// TIA Portal V18 export
// export: Created 2026-03-12T16:04:34.7244026Z, ExportSetting WithDefaults, DisplayName Totally Integrated Automation Portal, DisplayVersion V18 Update 5, DisplayName TIA Portal Openness, DisplayVersion V18 Update 5, DisplayName TIA Portal Version Control Interface, DisplayVersion V18, DisplayName SINAMICS Startdrive Advanced, DisplayVersion V18, DisplayName SINAMICS Startdrive G130, G150, S120, S150, SINAMICS MV, S210, DisplayVersion V18, DisplayName SINAMICS Startdrive G110M, G120, G120C, G120D, G120P, G115D, DisplayVersion V18, DisplayName STEP 7 Professional, DisplayVersion V18 Update 5, DisplayName STEP 7 Safety, DisplayVersion V18, DisplayName WinCC Professional, DisplayVersion V18 Update 5
FUNCTION_BLOCK "FB_HORÍMETROS"   // FB28, LAD
TITLE = Function Block HORÍMETRO - Contador de Horas
{ S7_Optimized_Access := 'TRUE' }
VERSION : 0.1
// Bloco para realizar a contagem de quantas horas cada motor/bomba passou ligado.
// stored: AutoNumber true, IsIECCheckEnabled false, IsRetainMemResEnabled false, MemoryReserve 100, SetENOAutomatically false, UDAEnableTagReadback false
   VAR_INPUT
      INPUT_BYTE : Byte;   // Entrada do sinal de falha instanciado na Network 1
   END_VAR
   VAR_IN_OUT
      HORIMETRO_1 : UInt;   // Saída do horímetro (horas trabalhadas da bomba)
      HORIMETRO_2 : UInt;
      HORIMETRO_3 : UInt;
      HORIMETRO_4 : UInt;
      HORIMETRO_5 : UInt;
      HORIMETRO_6 : UInt;
      HORIMETRO_7 : UInt;
      HORIMETRO_8 : UInt;
   END_VAR
   VAR
      Hor_1 : "FB_HORÍMETRO";
      Hor_2 { S7_SetPoint := 'True'} : "FB_HORÍMETRO";
      Hor_3 { S7_SetPoint := 'True'} : "FB_HORÍMETRO";
      Hor_4 { S7_SetPoint := 'True'} : "FB_HORÍMETRO";
      Hor_5 { S7_SetPoint := 'True'} : "FB_HORÍMETRO";
      Hor_6 { S7_SetPoint := 'True'} : "FB_HORÍMETRO";
      Hor_7 { S7_SetPoint := 'True'} : "FB_HORÍMETRO";
      Hor_8 { S7_SetPoint := 'True'} : "FB_HORÍMETRO";
   END_VAR
BEGIN

REGION Network 1
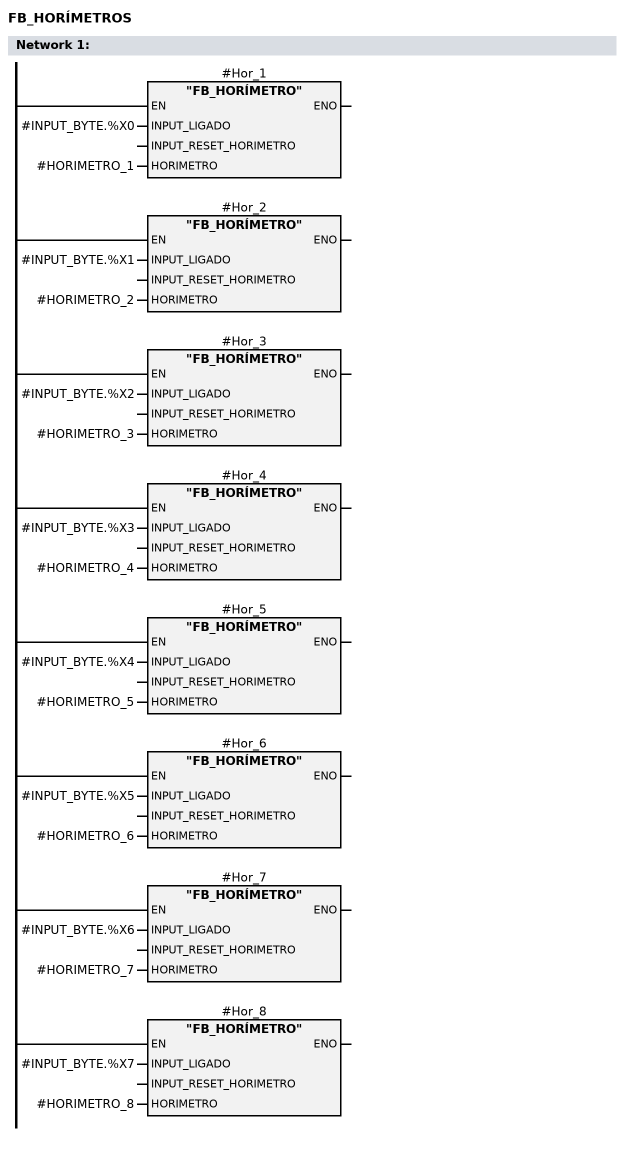
   RUNG wire#powerrail
      #Hor_1(INPUT_LIGADO := #INPUT_BYTE.%X0, INPUT_RESET_HORIMETRO :=, HORIMETRO := #HORIMETRO_1)
   END_RUNG
   RUNG wire#powerrail
      #Hor_2(INPUT_LIGADO := #INPUT_BYTE.%X1, INPUT_RESET_HORIMETRO :=, HORIMETRO := #HORIMETRO_2)
   END_RUNG
   RUNG wire#powerrail
      #Hor_3(INPUT_LIGADO := #INPUT_BYTE.%X2, INPUT_RESET_HORIMETRO :=, HORIMETRO := #HORIMETRO_3)
   END_RUNG
   RUNG wire#powerrail
      #Hor_4(INPUT_LIGADO := #INPUT_BYTE.%X3, INPUT_RESET_HORIMETRO :=, HORIMETRO := #HORIMETRO_4)
   END_RUNG
   RUNG wire#powerrail
      #Hor_5(INPUT_LIGADO := #INPUT_BYTE.%X4, INPUT_RESET_HORIMETRO :=, HORIMETRO := #HORIMETRO_5)
   END_RUNG
   RUNG wire#powerrail
      #Hor_6(INPUT_LIGADO := #INPUT_BYTE.%X5, INPUT_RESET_HORIMETRO :=, HORIMETRO := #HORIMETRO_6)
   END_RUNG
   RUNG wire#powerrail
      #Hor_7(INPUT_LIGADO := #INPUT_BYTE.%X6, INPUT_RESET_HORIMETRO :=, HORIMETRO := #HORIMETRO_7)
   END_RUNG
   RUNG wire#powerrail
      #Hor_8(INPUT_LIGADO := #INPUT_BYTE.%X7, INPUT_RESET_HORIMETRO :=, HORIMETRO := #HORIMETRO_8)
   END_RUNG
   // the same network as SCL:
   #Hor_1(INPUT_LIGADO := #INPUT_BYTE.%X0, HORIMETRO := #HORIMETRO_1);   // "FB_HORÍMETRO"
   #Hor_2(INPUT_LIGADO := #INPUT_BYTE.%X1, HORIMETRO := #HORIMETRO_2);   // "FB_HORÍMETRO"
   #Hor_3(INPUT_LIGADO := #INPUT_BYTE.%X2, HORIMETRO := #HORIMETRO_3);   // "FB_HORÍMETRO"
   #Hor_4(INPUT_LIGADO := #INPUT_BYTE.%X3, HORIMETRO := #HORIMETRO_4);   // "FB_HORÍMETRO"
   #Hor_5(INPUT_LIGADO := #INPUT_BYTE.%X4, HORIMETRO := #HORIMETRO_5);   // "FB_HORÍMETRO"
   #Hor_6(INPUT_LIGADO := #INPUT_BYTE.%X5, HORIMETRO := #HORIMETRO_6);   // "FB_HORÍMETRO"
   #Hor_7(INPUT_LIGADO := #INPUT_BYTE.%X6, HORIMETRO := #HORIMETRO_7);   // "FB_HORÍMETRO"
   #Hor_8(INPUT_LIGADO := #INPUT_BYTE.%X7, HORIMETRO := #HORIMETRO_8);   // "FB_HORÍMETRO"
END_REGION
END_FUNCTION_BLOCK
